# EPICS substitutions: siteApps/ICMP/icmpApp/Db/userHost.substitutions
# Example substitutions file

file "db/dbExample1.db" {
    { user = "ctrluserHost" }
}

file db/dbExample2.db {
    pattern { user, no, scan }
        { "ctrluserHost", 1, "1 second" }
        { "ctrluserHost", 2, "2 second" }
        { "ctrluserHost", 3, "5 second" }
}
